{attribute 'qualified_only'}
{attribute 'strict'}
{attribute 'to_string'}
TYPE E_CHECK_STATE :
(
  CHECK_INIT,
  AXIS_INDEX_OUT_OF_RANGE         :=  10,

	AXIS_REF_POINTER_INVALID        := 100,
  AXIS_CTRL_POINTER_INVALID,
  AXIS_STATE_POINTER_INVALID,
  AXIS_INFO_POINTER_INVALID,
  AXIS_DATA_POINTER_INVALID,
  AXIS_NC_PARAMETER_POINTER_INVALID,
  AXIS_HOME_PARAMETER_POINTER_INVALID,
  AXIS_GEAR_IN_PARAMETER_POINTER_INVALID,
  AXIS_GEAR_IN_MULTIMASTER_POINTER_INVALID,
  AXIS_MOTION_OPTIONS_POINTER_INVALID,

  NCI_NOT_ACTIVATED               := 200,
  NCI_CHANNEL_REF_POINTER_INVALID,
  NCI_AXIS_CONFIG_POINTER_INVALID,
  NCI_MCS_AXIS_POINTER_INVALID,
  NCI_AUX_AXIS_POINTER_INVALID,
  NCI_CTRL_POINTER_INVALID,
  NCI_STATE_POINTER_INVALID,
  NCI_R_PARAMETER_READ_POINTER_INVALID,
  NCI_R_PARAMETER_wRITE_POINTER_INVALID,
  NCI_M_FUNC_POINTER_INVALID,

  CAM_NOT_ACTIVATED               := 300,
  CAM_SLAVE_AXIS_REF_INVALID,
  CAM_SLAVE_ITF_MC_AXIS_INVALID,
  CAM_MASTER_AXIS_REF_INVALID,
  CAM_MOTION_FUNCTION_POINTER_INVALID,
  CAM_MOTION_FUNCTION_POINT_POINTER_INVALID,
  AXIS_LIMIT_SWITCHES_POINTER_INVALID,

  FLYING_SAW_NOT_ACTIVATED        := 400,
  FLYING_SLAVE_ITF_MC_AXIS_INVALID,
  FLYING_MASTER_AXIS_REF_INVALID,
  FLYING_FLY_DATA_POINTER_INVALID,
  FLYING_MOVE_DATA_POINTER_INVALID,
  FLYING_OPTIONS_POINTER_INVALID,
  FLYING_OPTIONS_SYNCMODE_SIZE_NOT_EQUAL,

  PARAMETER_SELECTOR              := 500,
  PARAMETER_SELECTOR_CTRL_REF_INVALID,
  PARAMETER_SELECTOR_STATE_REF_INVALID,
  PARAMETER_SELECTOR_AXIS_ITF_INVALID,


  CHECK_DONE                      := 10000
  
)UINT;
END_TYPE

(* stored: Version 1.1.0.1, ProductVersion 3.1.4026.18
   DUT E_CHECK_STATE: Id {1ade6feb-94c7-01c0-0791-138199d866b6} *)
